PROGRAM MAIN
VAR
END_VAR

//SavePersistentVariables();

END_PROGRAM

(* stored: Version 1.1.0.1, ProductVersion 3.1.4020.12
   POU MAIN: Id {89a4b85f-5d38-482c-b479-b96ffddc6afa}, SpecialFunc None *)
